{attribute 'qualified_only'}
{attribute 'strict'}
TYPE CoffeType :
(
	Cappucciono 		:= 1,
	Caffelatte 			:= 2,
	Latte				:= 3,
	FlatWhite			:= 4,
	SingleES			:= 5,
	DoubleES			:= 6,
	Milk				:= 7
);
END_TYPE

(* stored: Version 1.1.0.1, ProductVersion 3.1.4024.12
   DUT CoffeType: Id {66ff464d-bfbf-46b6-8616-303cfaea57da} *)
